(* CoDeSys 2.3 export: CODESYSEXPORT22_2.EXP *)

(* POU MAIN, ST *)
PROGRAM MAIN
(*Main program for application. Uses PackML state model to control the execution of the application*)
VAR
	tonStarting				: TON;
	rsEmergencyClear	: RS;	(*RS - flip-flop for Emergency clear info*)
END_VAR
(* ****** Section 1: Initialisations and default values. Initial conditions for variables on every PLC cycle*)
(*Default values*)
fbStateModel.bSC := FALSE;
(*System resets*)

(* ****** Section 2: Actions in your program without considering the Control Mode. I.e. actions are performed same way indenpendent on
current Control Mode selection.*)
(*Mode independent state actions. Change / Add / Remove states according your need*)
CASE fbStateModel.eState OF
eSt_Aborting:
	(* One can make specific actions in case of specific Mode-State combination.
	   One can also consider to call a specific program when in specific Mode-State combination*)
	actAborting;
	fbStateModel.bSC := TRUE;		(*MODIFY*)
eSt_Clearing:
	fbStateModel.bSC := TRUE;		(*MODIFY*)
eSt_Resetting:
	fbStateModel.bSC := TRUE;
eSt_Holding:
	fbStateModel.bSC := TRUE;		(*MODIFY*)
eSt_UnHolding:
	fbStateModel.bSC := TRUE;		(*MODIFY*)
eSt_Suspending:
	fbStateModel.bSC := TRUE;		(*MODIFY*)
eSt_Unsuspending:
	fbStateModel.bSC := TRUE;		(*MODIFY*)
END_CASE;

(* ****** Section 3: Actions in your program which are Control Mode specific. Two nested case structures where outer one selects the
control mode and inner the PackML state. In order to avoid conflicts, it would be better to process each PackML state either in Section 2 
or Section 3, but not in both. *)
(*Execution mode related state actions. Change / Add / Remove mode and states according your need*)
CASE fbStateModel.eMode OF
(*MODE: MANUAL*)
eMode_Manual:
	(* ****** Section 3.1: PackML state based processing actions when Control Mode is Manual.*)
	CASE fbStateModel.eState OF
	eSt_Starting:
		IF IPressureApplied THEN
			fbStateModel.bSC := TRUE;			(*MODIFY*)
		END_IF
	eSt_Stopping:
		fbStateModel.bSC := TRUE;			(*MODIFY*)
	END_CASE;

(*MODE: AUTOMATIC*)
eMode_Automatic:
	(* ****** Section 3.2: PackML state based processing actions when Control Mode is Automatic.*)
	CASE fbStateModel.eState OF
	eSt_Idle:
		tonStarting(IN:=FALSE , PT:= , Q=> , ET=> );	(*MODIFY*)
	eSt_Starting:
		(* tonStarting(IN:=TRUE , PT:=T#2s , Q=> , ET=> );
		fbStateModel.bSC := tonStarting.Q; *)
		IF IPressureApplied THEN
			bDriveEnabled := TRUE;
			PRG_Initialisation(bReset:= , bExecute:= TRUE , bDone=> );
		END_IF

		IF PRG_Initialisation.bDone THEN
			PRG_Initialisation(bReset:= , bExecute:= FALSE , bDone=> );
			fbStateModel.bSC := TRUE;
		END_IF
	eSt_Completing:
		fbStateModel.bSC := TRUE;					(*MODIFY*)
	eSt_Completed:
		;
	END_CASE;

(* ****** Section 4: Grouping PackML states for calling Programs or FB instances.
This is to avoid repetition inside above case structure in Section 3. With IF clause setting lower (and upper) state limits we can filter out the states when we want to call 
specific programs. The order of states is defined in Tab:Data types > E_PackMLState. eSt_Aborting is lowest and eSt_Completed is highest.
Here we filter calling programs, only when we are in higher states than Stopped. 
This can be pulled out as completely separated section, like in PackML_StateModel_v2-2.pro project. There is inside IF again CASE which process each Control Mode separately.*)
(*Execution part. Making calls for program if we are on states above Stopped*)
	(*If we are between specific states, make some action or program call*)
	IF  (fbStateModel.eState>eSt_Starting) AND (fbStateModel.eState<=eSt_Completing) THEN
		(*Make here the actions / calls Good place to start with is PRG_Sorting (PRG)*)
		PRG_AutoSort(bExecute:= TRUE , bReset:= , bDone=> , bStopOk=> );
	END_IF;

(*MODE: UNKNOWN*)
ELSE	(*Error*)
	; (*TODO*)
END_CASE;

(* ****** Section 5: Calling the fbStateModel instance.
Here the instance of state model is called and all triggering inputs are set, but bSC (State Completed), which you control in your programs. 
This is indication that your program has  finished certain stage.
- Pay attention where the instance fbStateModel is defined. Do you do it in global variables or e.g. here in PRG_MAIN? Important is to use the 
same instance in all places, so that machine state is unique and shared. Remember, if you have multiple definitions, the PRG_MAIN "hides" 
the global one, and might lead to problems elswhere, when you think you are using the same instance, but actually are not. 
- In case you are using the PackML visualisation (VC_PackMLStates), make sure you connect its placeholder to the very same PackML FB instance.
- The Mask for wIgnoreState is created as following. I use binary base for the value(2#). The lowest bit in the mask corresponds the eSt_Aborting
 in E_PackMLState. The next is eSt_Aborted, and so on. Specific state is ignored and jumped over when it is masked out i.e. ignored by having 1 
in that position. Note that implementation allows this only for selected states. See FB_PackMLStateModel_ST code for further details.*)
(*Calling & Updating the state model*)
(*TODO: Evaluate and change all input conditions according your application needs*)
fbStateModel(
	bResetFB:= ,
	eModeReq:= HMI_uModeReq,
	wIgnoreState := 2#000000,		(*TODO: Which states should be ignodered. Default: 2#000000 or 2#100000. The latter is ignoring Resetting state*)
	bSC:= ,			(*Must not be assigned ANY variable, because fb input is directly operated!!!*)
	bAbort:= NOT (IEmergencyClear  OR  IPressureApplied),
	bClear:= IEmergencyClear,
	bReset:= I_Btn_Start,
	bStart:= I_Btn_Start,
	bHold:= ,
	bUn_Hold:= ,
	bSuspend:= ,
	bUn_Suspend:= ,
	bStop:= I_Btn_Stop ,
	bComplete:= ,
	bAck_Completed:= ,
	eMode=> PLC_uModeCurrent,
	eState=> PLC_uStateCurrent);

(* ****** Section 6: Here we update all outputs according the current state of our PackML model. This allows us to process the in single location.
The control of outputs is bind to state, not e.g. to inputs. The inputs are the one driving the PackML model forward. Again CASE structure can be used.*)
(*Call for HMI and UI update*)
(*PRG_Drive_Link()*);
HMI_and_UI_Update;
END_PROGRAM
ACTION actAborting:
bDriveEnabled := FALSE;
PRG_Sorting(bReset:=TRUE , bExecute:= FALSE);
END_ACTION
ACTION HMI_and_UI_Update:
(*Simulate emergency stop circuitry*)
rsEmergencyClear(
	SET:= I_Btn_Reset,
	RESET1:= I_Btn_EStop ,
	Q1=> IEmergencyClear);

(*HMI Update*)
PRG_Blinking (bSign4Hz=> , bSign2Hz=> , bSign1Hz=> , bSign0_5Hz=> );
(*Init values*)
O_Light_BeaconRed := FALSE;

(*OLight_Start :=  (fbStateModel.eState >= eSt_Resetting) AND (fbStateModel.eState < eSt_Completed);*)
CASE fbStateModel.eState OF
eSt_Aborting, eSt_Aborted:
	O_Light_BeaconRed := PRG_Blinking.bSign1Hz;
eSt_Clearing:
	O_Light_BeaconRed := PRG_Blinking.bSign0_5Hz;
eSt_Stopped, eSt_Completed:
	O_Light_BeaconRed := TRUE;
eSt_Starting:
	;
END_CASE;
END_ACTION

(* POU Programs/PRG_Initialisation, SFC *)
PROGRAM PRG_Initialisation
(*Template program for system initialisation*)
VAR_INPUT
	bReset	: BOOL := FALSE;	(*Reseting the SFC*)
	bExecute	: BOOL;			(*Executes PRG*)
END_VAR
VAR_OUTPUT
	bDone		: BOOL;		(*Program operations done*)
END_VAR
VAR
(* -------------INTERNAL-------------------*)
	tonMoveDelay		: TON;
	tMoveDelay		: TIME := T#1s;
	bInitDone			: BOOL:=FALSE;	(*Initialisation done*)
	bGatesClosed	: BOOL:=FALSE;	(*Initialisation done*)
	bActuRetracted	: BOOL:=FALSE;
	bDriveAtLoading	: BOOL:=FALSE;

(*System variables. See SFC-flags: http://infosys.beckhoff.com/content/1033/tcplccontrol/html/tcplcctrl_editorsfc.htm?id=24319#SFC-Flags*)
	SFCReset		: BOOL := FALSE;	(*For reseting the SFC*)
END_VAR
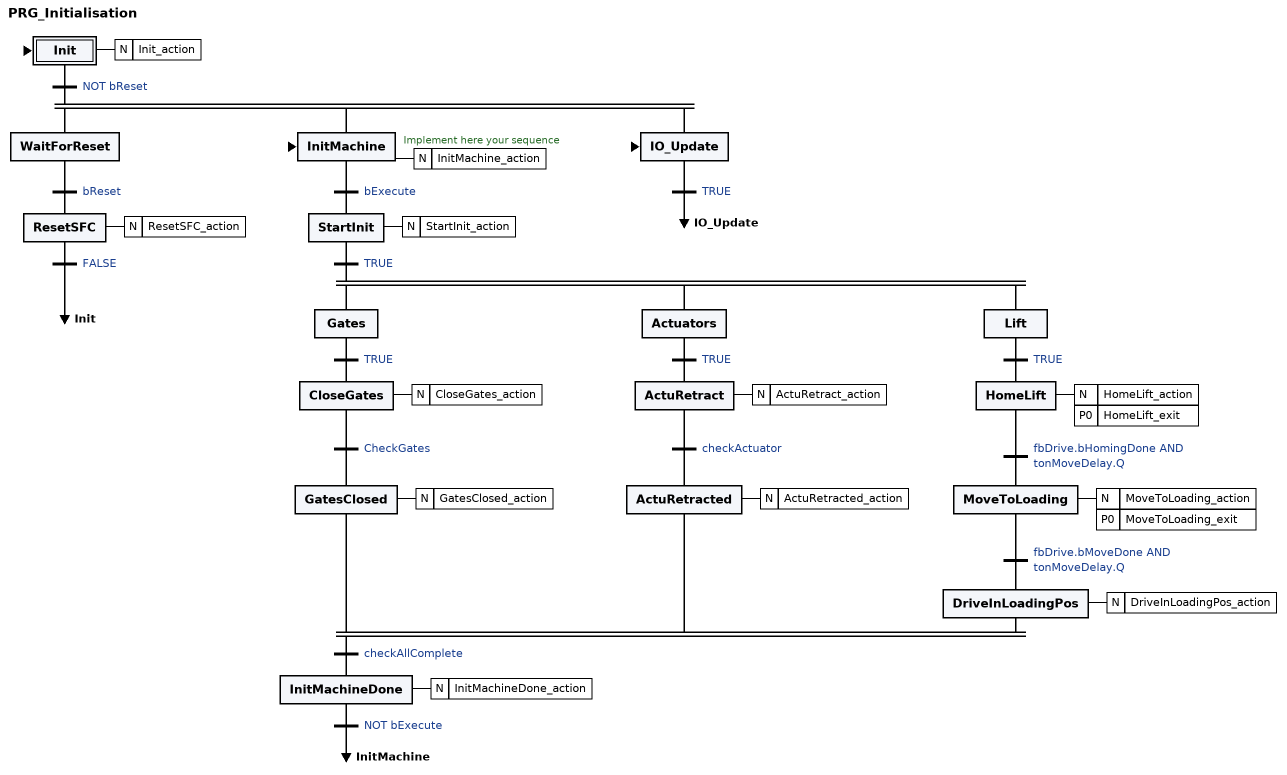
INITIAL_STEP Init:
	Init_action(N);
END_STEP
TRANSITION FROM Init TO (WaitForReset, InitMachine, IO_Update) := NOT bReset;
END_TRANSITION
STEP WaitForReset:
END_STEP
TRANSITION FROM WaitForReset TO ResetSFC := bReset;
END_TRANSITION
STEP ResetSFC:
	ResetSFC_action(N);
END_STEP
TRANSITION FROM ResetSFC TO Init := FALSE;
END_TRANSITION
STEP InitMachine: (* Implement here your sequence *)
	InitMachine_action(N);
END_STEP
TRANSITION FROM InitMachine TO StartInit := bExecute;
END_TRANSITION
STEP StartInit:
	StartInit_action(N);
END_STEP
TRANSITION FROM StartInit TO (Gates, Actuators, Lift) := TRUE;
END_TRANSITION
STEP Gates:
END_STEP
TRANSITION FROM Gates TO CloseGates := TRUE;
END_TRANSITION
STEP CloseGates:
	CloseGates_action(N);
END_STEP
TRANSITION FROM CloseGates TO GatesClosed := CheckGates;
END_TRANSITION
STEP GatesClosed:
	GatesClosed_action(N);
END_STEP
STEP Actuators:
END_STEP
TRANSITION FROM Actuators TO ActuRetract := TRUE;
END_TRANSITION
STEP ActuRetract:
	ActuRetract_action(N);
END_STEP
TRANSITION FROM ActuRetract TO ActuRetracted := checkActuator;
END_TRANSITION
STEP ActuRetracted:
	ActuRetracted_action(N);
END_STEP
STEP Lift:
END_STEP
TRANSITION FROM Lift TO HomeLift := TRUE;
END_TRANSITION
STEP HomeLift:
	HomeLift_action(N);
	HomeLift_exit(P0);
END_STEP
TRANSITION FROM HomeLift TO MoveToLoading := fbDrive.bHomingDone AND tonMoveDelay.Q;
END_TRANSITION
STEP MoveToLoading:
	MoveToLoading_action(N);
	MoveToLoading_exit(P0);
END_STEP
TRANSITION FROM MoveToLoading TO DriveInLoadingPos := fbDrive.bMoveDone AND tonMoveDelay.Q;
END_TRANSITION
STEP DriveInLoadingPos:
	DriveInLoadingPos_action(N);
END_STEP
TRANSITION FROM (GatesClosed, ActuRetracted, DriveInLoadingPos) TO InitMachineDone := checkAllComplete;
END_TRANSITION
STEP InitMachineDone:
	InitMachineDone_action(N);
END_STEP
TRANSITION FROM InitMachineDone TO InitMachine := NOT bExecute;
END_TRANSITION
STEP IO_Update:
END_STEP
TRANSITION FROM IO_Update TO IO_Update := TRUE;
END_TRANSITION

ACTION Init_action:
(*Clear Reset SFC*)
SFCReset:= FALSE;
bDone := FALSE;
END_ACTION

ACTION ResetSFC_action:
(*Reset SFC*)
SFCReset:=TRUE;
END_ACTION

ACTION InitMachine_action:
(*Do some actions...

Sulje kaikki portit ... JA tarkista Steppiä seuraavassa transitioehdossa, että kaikki portit ovat kiinni
Close all gates.... and check in following transition that ALL gates are closed*)

;
END_ACTION

ACTION StartInit_action:
bDone := FALSE;
END_ACTION

ACTION CloseGates_action:
OGateUp		:= FALSE;
OGateMid		:= FALSE;
OGateLow		:= FALSE;
OSorterGate	:= FALSE;
END_ACTION

ACTION GatesClosed_action:
bGatesClosed := TRUE;
END_ACTION

ACTION ActuRetract_action:
OSorterLift	 := FALSE;
OEjector	 := FALSE;
END_ACTION

ACTION ActuRetracted_action:
bActuRetracted := TRUE;
END_ACTION

ACTION HomeLift_action:
fbDrive.bStart := TRUE;
tonMoveDelay(IN:=TRUE , PT:= tMoveDelay);
END_ACTION

ACTION HomeLift_exit:
fbDrive.bStart:= FALSE;
tonMoveDelay(IN:=FALSE);
END_ACTION

ACTION MoveToLoading_action:
fbDrive.wTarget := GPOS_LOADING;
fbDrive.bStart:= TRUE;
tonMoveDelay(IN:=TRUE , PT:= tMoveDelay);
END_ACTION

ACTION MoveToLoading_exit:
fbDrive.bStart:= FALSE;
tonMoveDelay(IN:=FALSE);
END_ACTION

ACTION DriveInLoadingPos_action:
bDriveAtLoading := TRUE;
END_ACTION

ACTION InitMachineDone_action:
bDone := TRUE;
END_ACTION

TRANSITION CheckGates:
_FBD_ (* Function Block Diagram *)
NETWORK 1
	AND(IGateClosedUp, IGateClosedMid, IGateClosedLow, ISorterGateClosed)
_END_FBD_
END_TRANSITION

TRANSITION checkActuator:
_FBD_ (* Function Block Diagram *)
NETWORK 1
	AND(ISorterLiftDown, NOT OEjector)
_END_FBD_
END_TRANSITION

TRANSITION checkAllComplete:
_FBD_ (* Function Block Diagram *)
NETWORK 1
	AND(bGatesClosed, bActuRetracted, bDriveAtLoading)
_END_FBD_
END_TRANSITION
END_PROGRAM

(* POU Programs/PRG_AutoSort, ST *)
PROGRAM PRG_AutoSort
VAR_INPUT
	bExecute	: BOOL;
	bReset	: BOOL := FALSE;
END_VAR
VAR_OUTPUT
	bDone		: BOOL;		(*Program operations done*)
	bStopOk    : BOOL;
END_VAR
VAR
	fbSorter	: FB_Sorter;
	fbLift		: FB_Lift;
	bBatchComplete  : BOOL := FALSE;
END_VAR
actUpdateIO;
actCheckAllOkStop;

CASE fbStateModel.eState OF
	eSt_Idle:
		fbStateModel.bComplete  := FALSE;
		fbStateModel.bSC 		:= TRUE;
	eSt_Resetting:
		fbStateModel.bSC := TRUE;
	eSt_Stopping:
		fbStateModel.bStop := FALSE;

		IF  bStopOk THEN
			fbStateModel.bSC := TRUE;
		END_IF
	eSt_Execute:
		fbSorter (bEnable :=  TRUE , bReset := FALSE);
		fbLift(bEnable :=  TRUE , bReset := FALSE);
		IF bBatchComplete  THEN
			fbStateModel.bComplete := TRUE;
		END_IF

	eSt_Completing:
		fbStateModel.bComplete := FALSE;
		IF bStopOK THEN
			fbStateModel.bSC := TRUE;
		END_IF

	eSt_Unsuspending:
		fbStateModel.bSC := TRUE;

	eSt_Suspending:
		fbStateModel.bSuspend := FALSE;
		fbStateModel.bSC := TRUE;

END_CASE
END_PROGRAM
ACTION actCheckAllOKStop:
IF fbSorter.bStopOK AND  fbLift.bStopOK THEN
	bStopOK := TRUE;
ELSE
	bStopOK := FALSE;
END_IF
END_ACTION
ACTION actUpdateIO:
fbSorter (
	bReset:= ,
	bEnable:= bExecute,
	I_SensorOpt:= ISensorOpt ,
	I_SensorInd:= ISensorInd,
	I_SorterLiftUp:= ISorterLiftUp ,
	I_SorterLiftDown:= ISorterLiftDown,
	hiRdyToReceive_FromDS:= fbLift.hoReadyToRecieve_ToUS ,
	hiBallAvail_FromUS:= ,
	bStopOK=> ,
	bBallLoaded=> ,
	bCurBallMetal=> ,
	O_SorterGate=> OSorterGate ,
	O_SorterLift=> OSorterLift ,
	hoBallAvail_ToDS=> ,
	hoReadyToRecieve_ToUS=> );

fbLift (
	bReset:= ,
	bEnable:= bExecute,
	I_LimitUp:= ILimitUp  ,
	I_LimitLow:= ILimitLow,
	I_WaitingBallMetal:= fbSorter.bCurBallMetal  ,
	I_SenColourYellow:= ISenColourYellow ,
	I_SenColourBlue:= ISenColourBlue ,
	I_SenColourGreen:= ISenColourGreen,
	I_SenColourRed:= ISenColourRed ,
	hiRdyToReceive_FromDS:= ,
	hiBallAvail_FromUS:= fbSorter.hoBallAvail_ToDS ,
	bStopOK=> ,
	bBallLoaded=> , 
	bCurBallMetal=> , 
	O_Ejector=> OEjector ,
	hoBallAvail_ToDS=> , 
	hoReadyToRecieve_ToUS=> );
END_ACTION

(* POU FBs/FB_Sorter, SFC *)
FUNCTION_BLOCK FB_Sorter
VAR_INPUT
	bReset			: BOOL;	(*Reset Request*)
	bEnable			: BOOL;
	I_SensorOpt		: BOOL;
	I_SensorInd		: BOOL;
	I_SorterLiftUp		: BOOL;
	I_SorterLiftDown	: BOOL;

	(*SMEMA Handshake Inputs*)
	hiRdyToReceive_FromDS	: BOOL;
	hiBallAvail_FromUS			: BOOL;
END_VAR
VAR_OUTPUT
	bStopOK			: BOOL;
	bBallLoaded		: BOOL;
	bCurBallMetal		: BOOL;
	O_SorterGate		: BOOL;
	O_SorterLift		: BOOL;

	(*SMEMA Handshake Outputs*)
	hoBallAvail_ToDS				: BOOL;
	hoReadyToRecieve_ToUS	: BOOL;
END_VAR
VAR
	tTransferDelay: TIME := T#4s;
	tMoveDelay	: TIME := T#2s;
	fbDelay		: FB_Wait;
	bLocalReset	: BOOL;	(*Performs local reset*)
	SFCReset 	: BOOL;	(*Resets the execution of SFC to init once this SFCFlag is set true *)
END_VAR
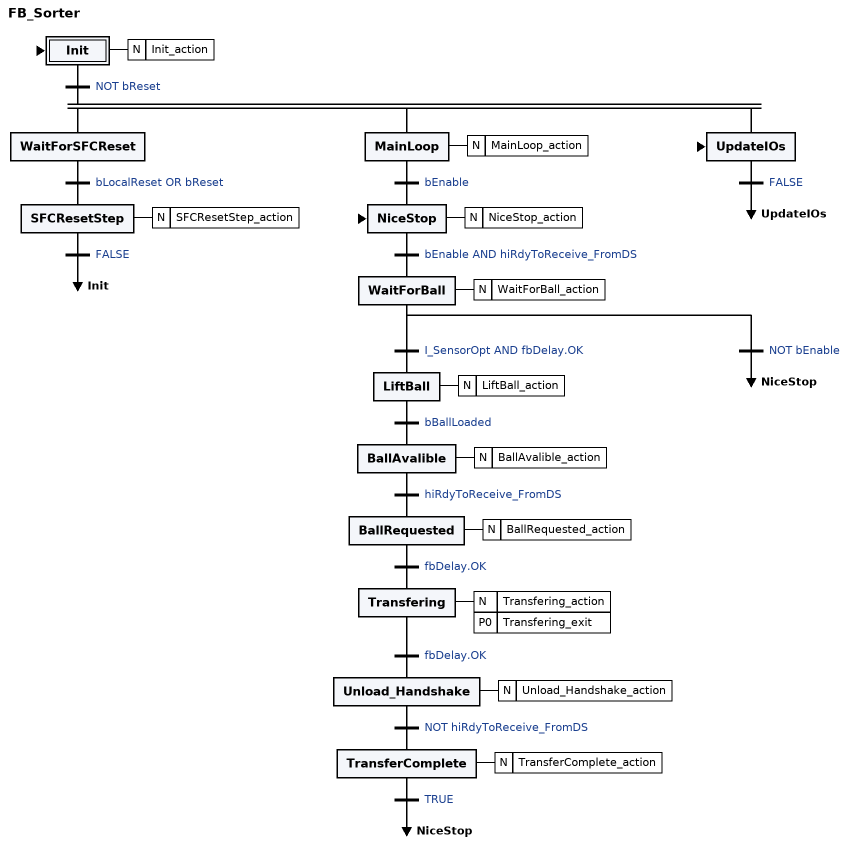
INITIAL_STEP Init:
	Init_action(N);
END_STEP
TRANSITION FROM Init TO (WaitForSFCReset, MainLoop, UpdateIOs) := NOT bReset;
END_TRANSITION
STEP WaitForSFCReset:
END_STEP
TRANSITION FROM WaitForSFCReset TO SFCResetStep := bLocalReset OR bReset;
END_TRANSITION
STEP MainLoop:
	MainLoop_action(N);
END_STEP
TRANSITION FROM MainLoop TO NiceStop := bEnable;
END_TRANSITION
STEP NiceStop:
	NiceStop_action(N);
END_STEP
TRANSITION FROM NiceStop TO WaitForBall := bEnable AND hiRdyToReceive_FromDS;
END_TRANSITION
STEP WaitForBall:
	WaitForBall_action(N);
END_STEP
TRANSITION FROM WaitForBall TO LiftBall := I_SensorOpt AND fbDelay.OK;
END_TRANSITION
TRANSITION FROM WaitForBall TO NiceStop := NOT bEnable;
END_TRANSITION
STEP LiftBall:
	LiftBall_action(N);
END_STEP
TRANSITION FROM LiftBall TO BallAvalible := bBallLoaded;
END_TRANSITION
STEP BallAvalible:
	BallAvalible_action(N);
END_STEP
TRANSITION FROM BallAvalible TO BallRequested := hiRdyToReceive_FromDS;
END_TRANSITION
STEP BallRequested:
	BallRequested_action(N);
END_STEP
TRANSITION FROM BallRequested TO Transfering := fbDelay.OK;
END_TRANSITION
STEP Transfering:
	Transfering_action(N);
	Transfering_exit(P0);
END_STEP
TRANSITION FROM Transfering TO Unload_Handshake := fbDelay.OK;
END_TRANSITION
STEP Unload_Handshake:
	Unload_Handshake_action(N);
END_STEP
TRANSITION FROM Unload_Handshake TO TransferComplete := NOT hiRdyToReceive_FromDS;
END_TRANSITION
STEP TransferComplete:
	TransferComplete_action(N);
END_STEP
TRANSITION FROM TransferComplete TO NiceStop := TRUE;
END_TRANSITION
STEP UpdateIOs:
END_STEP
TRANSITION FROM UpdateIOs TO UpdateIOs := FALSE;
END_TRANSITION
STEP SFCResetStep:
	SFCResetStep_action(N);
END_STEP
TRANSITION FROM SFCResetStep TO Init := FALSE;
END_TRANSITION

ACTION Init_action:
SFCReset := FALSE;
bLocalReset	:= FALSE;
bStopOK := FALSE;
END_ACTION

ACTION MainLoop_action:
hoBallAvail_ToDS			  := FALSE;
hoReadyToRecieve_ToUS := FALSE;
END_ACTION

ACTION NiceStop_action:
bBallLoaded 				  := FALSE;
bStopOK					  := TRUE;
hoBallAvail_ToDS			  := FALSE;
hoReadyToRecieve_ToUS := FALSE;
END_ACTION

ACTION WaitForBall_action:
fbDelay(IN_TIME:=tMoveDelay);
(* Move Lift Down *)
O_SorterLift := FALSE;
END_ACTION

ACTION LiftBall_action:
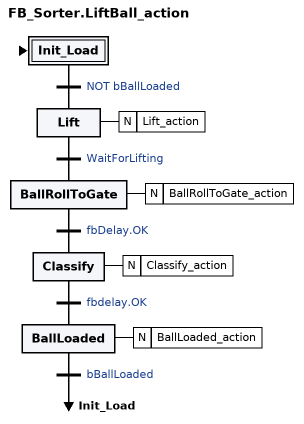
INITIAL_STEP Init_Load:
END_STEP
TRANSITION FROM Init_Load TO Lift := NOT bBallLoaded;
END_TRANSITION
STEP Lift:
	Lift_action(N);
END_STEP
TRANSITION FROM Lift TO BallRollToGate := WaitForLifting;
END_TRANSITION
STEP BallRollToGate:
	BallRollToGate_action(N);
END_STEP
TRANSITION FROM BallRollToGate TO Classify := fbDelay.OK;
END_TRANSITION
STEP Classify:
	Classify_action(N);
END_STEP
TRANSITION FROM Classify TO BallLoaded := fbdelay.OK;
END_TRANSITION
STEP BallLoaded:
	BallLoaded_action(N);
END_STEP
TRANSITION FROM BallLoaded TO Init_Load := bBallLoaded;
END_TRANSITION

ACTION Lift_action:
O_SorterLift := TRUE;
fbDelay(IN_TIME:=tMoveDelay);
END_ACTION

ACTION BallRollToGate_action:
fbDelay(IN_TIME:=tMoveDelay);
END_ACTION

ACTION Classify_action:
fbDelay(IN_TIME:=tMoveDelay);
IF I_SensorInd THEN
	bCurBallMetal := FALSE;
ELSE
	bCurBallMetal := TRUE;
END_IF
END_ACTION

ACTION BallLoaded_action:
bBallLoaded := TRUE;
END_ACTION

TRANSITION WaitForLifting:
_FBD_ (* Function Block Diagram *)
NETWORK 1
	AND(I_SorterLiftUp, fbDelay.OK, NOT I_SensorOpt)
_END_FBD_
END_TRANSITION
END_ACTION

ACTION BallAvalible_action:
hoBallAvail_ToDS := TRUE;
END_ACTION

ACTION BallRequested_action:
fbDelay(IN_TIME:=tMoveDelay);
END_ACTION

ACTION Transfering_action:
O_SorterGate := TRUE;
fbDelay(IN_TIME:=tTransferDelay);
END_ACTION

ACTION Transfering_exit:
O_SorterGate := FALSE;
END_ACTION

ACTION Unload_Handshake_action:
hoBallAvail_ToDS := FALSE;
END_ACTION

ACTION TransferComplete_action:
bBallLoaded := FALSE;
END_ACTION

ACTION SFCResetStep_action:
SFCReset := TRUE;
END_ACTION
END_FUNCTION_BLOCK

(* POU FBs/FB_Lift, SFC *)
FUNCTION_BLOCK FB_Lift
VAR_INPUT
	bReset			 : BOOL;	(*Reset Request*)
	bEnable			 : BOOL;
	I_LimitUp 			 : BOOL;
	I_LimitLow 	        : BOOL;
	I_WaitingBallMetal : BOOL;

	(* ColourSensor *)
	I_SenColourYellow		:BOOL;	(*Colour sensor In1 - Yellow*)
	I_SenColourBlue		:BOOL;	(*Colour sensor In2 - Blue*)
	I_SenColourGreen		:BOOL;	(*Colour sensor In3 - Green*)
	I_SenColourRed		:BOOL;	(*Colour sensor In4 - Red*)

	(*SMEMA Handshake Inputs*)
	hiRdyToReceive_FromDS	: BOOL;
	hiBallAvail_FromUS			: BOOL;
END_VAR
VAR_OUTPUT
	bStopOK		: BOOL;
	bBallLoaded	: BOOL;
	bCurBallMetal	: BOOL;
	bCurrentBall 	: E_BallColour := NoColour;

	O_Ejector		:BOOL;

	(*SMEMA Handshake Outputs*)
	hoBallAvail_ToDS				: BOOL;
	hoReadyToRecieve_ToUS	: BOOL;
END_VAR
VAR
	bBallRequested : BOOL := FALSE;
	fbTransferBall	:FB_TransferBall;

	fbDelay		: FB_Wait;
	tonMoveDelay	: TON;
	tonSensorDelay	: TON;
	tTransferDelay: TIME := T#4s;
	tMoveDelay	: TIME := T#4s;
	tSensorDelay	: TIME := T#2s;
	bLocalReset	: BOOL;	(*Performs local reset*)
	SFCReset 	: BOOL;	(*Resets the execution of SFC to init once this SFCFlag is set true *)
END_VAR
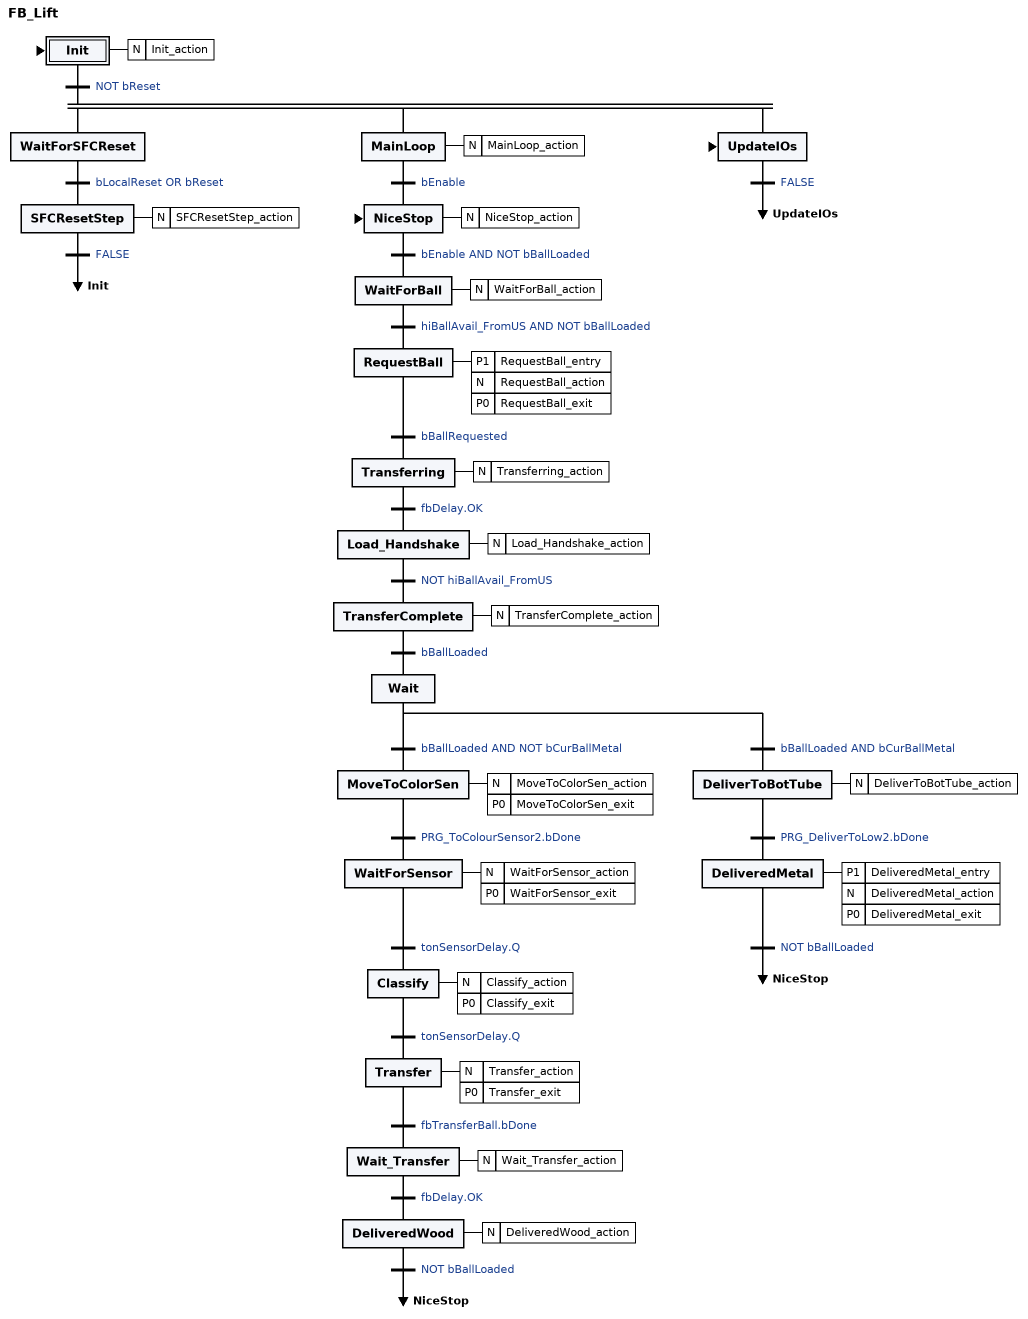
INITIAL_STEP Init:
	Init_action(N);
END_STEP
TRANSITION FROM Init TO (WaitForSFCReset, MainLoop, UpdateIOs) := NOT bReset;
END_TRANSITION
STEP WaitForSFCReset:
END_STEP
TRANSITION FROM WaitForSFCReset TO SFCResetStep := bLocalReset OR bReset;
END_TRANSITION
STEP MainLoop:
	MainLoop_action(N);
END_STEP
TRANSITION FROM MainLoop TO NiceStop := bEnable;
END_TRANSITION
STEP NiceStop:
	NiceStop_action(N);
END_STEP
TRANSITION FROM NiceStop TO WaitForBall := bEnable AND NOT bBallLoaded;
END_TRANSITION
STEP WaitForBall:
	WaitForBall_action(N);
END_STEP
TRANSITION FROM WaitForBall TO RequestBall := hiBallAvail_FromUS AND NOT bBallLoaded;
END_TRANSITION
STEP RequestBall:
	RequestBall_entry(P1);
	RequestBall_action(N);
	RequestBall_exit(P0);
END_STEP
TRANSITION FROM RequestBall TO Transferring := bBallRequested;
END_TRANSITION
STEP Transferring:
	Transferring_action(N);
END_STEP
TRANSITION FROM Transferring TO Load_Handshake := fbDelay.OK;
END_TRANSITION
STEP Load_Handshake:
	Load_Handshake_action(N);
END_STEP
TRANSITION FROM Load_Handshake TO TransferComplete := NOT hiBallAvail_FromUS;
END_TRANSITION
STEP TransferComplete:
	TransferComplete_action(N);
END_STEP
TRANSITION FROM TransferComplete TO Wait := bBallLoaded;
END_TRANSITION
STEP Wait:
END_STEP
TRANSITION FROM Wait TO MoveToColorSen := bBallLoaded AND NOT bCurBallMetal;
END_TRANSITION
TRANSITION FROM Wait TO DeliverToBotTube := bBallLoaded AND bCurBallMetal;
END_TRANSITION
STEP MoveToColorSen:
	MoveToColorSen_action(N);
	MoveToColorSen_exit(P0);
END_STEP
TRANSITION FROM MoveToColorSen TO WaitForSensor := PRG_ToColourSensor2.bDone;
END_TRANSITION
STEP WaitForSensor:
	WaitForSensor_action(N);
	WaitForSensor_exit(P0);
END_STEP
TRANSITION FROM WaitForSensor TO Classify := tonSensorDelay.Q;
END_TRANSITION
STEP Classify:
	Classify_action(N);
	Classify_exit(P0);
END_STEP
TRANSITION FROM Classify TO Transfer := tonSensorDelay.Q;
END_TRANSITION
STEP Transfer:
	Transfer_action(N);
	Transfer_exit(P0);
END_STEP
TRANSITION FROM Transfer TO Wait_Transfer := fbTransferBall.bDone;
END_TRANSITION
STEP Wait_Transfer:
	Wait_Transfer_action(N);
END_STEP
TRANSITION FROM Wait_Transfer TO DeliveredWood := fbDelay.OK;
END_TRANSITION
STEP DeliveredWood:
	DeliveredWood_action(N);
END_STEP
TRANSITION FROM DeliveredWood TO NiceStop := NOT bBallLoaded;
END_TRANSITION
STEP DeliverToBotTube:
	DeliverToBotTube_action(N);
END_STEP
TRANSITION FROM DeliverToBotTube TO DeliveredMetal := PRG_DeliverToLow2.bDone;
END_TRANSITION
STEP DeliveredMetal:
	DeliveredMetal_entry(P1);
	DeliveredMetal_action(N);
	DeliveredMetal_exit(P0);
END_STEP
TRANSITION FROM DeliveredMetal TO NiceStop := NOT bBallLoaded;
END_TRANSITION
STEP UpdateIOs:
END_STEP
TRANSITION FROM UpdateIOs TO UpdateIOs := FALSE;
END_TRANSITION
STEP SFCResetStep:
	SFCResetStep_action(N);
END_STEP
TRANSITION FROM SFCResetStep TO Init := FALSE;
END_TRANSITION

ACTION Init_action:
SFCReset := FALSE;
bLocalReset	:= FALSE;
END_ACTION

ACTION MainLoop_action:
hoBallAvail_ToDS			  := FALSE;
hoReadyToRecieve_ToUS := FALSE;
END_ACTION

ACTION NiceStop_action:
bStopOK	  	:= TRUE;
bCurrentBall	:= NoColour;
END_ACTION

ACTION WaitForBall_action:
bBallLoaded := FALSE;
hoReadyToRecieve_ToUS := TRUE;
END_ACTION

ACTION RequestBall_entry:
bStopOK := FALSE;
END_ACTION

ACTION RequestBall_action:
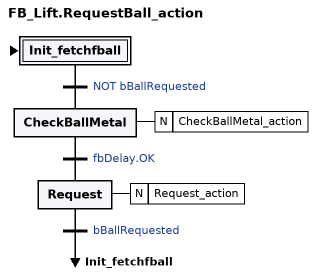
INITIAL_STEP Init_fetchfball:
END_STEP
TRANSITION FROM Init_fetchfball TO CheckBallMetal := NOT bBallRequested;
END_TRANSITION
STEP CheckBallMetal:
	CheckBallMetal_action(N);
END_STEP
TRANSITION FROM CheckBallMetal TO Request := fbDelay.OK;
END_TRANSITION
STEP Request:
	Request_action(N);
END_STEP
TRANSITION FROM Request TO Init_fetchfball := bBallRequested;
END_TRANSITION

ACTION CheckBallMetal_action:
bCurBallMetal	 := I_WaitingBallMetal;
fbDelay(IN_TIME:=T#2s);
END_ACTION

ACTION Request_action:
hoReadyToRecieve_ToUS := TRUE;
bBallRequested := TRUE;
END_ACTION
END_ACTION

ACTION RequestBall_exit:
bBallRequested := FALSE;
END_ACTION

ACTION Transferring_action:
fbDelay(IN_TIME:=tTransferDelay);
END_ACTION

ACTION Load_Handshake_action:
hoReadyToRecieve_ToUS := FALSE;
END_ACTION

ACTION TransferComplete_action:
bBallLoaded := TRUE;
END_ACTION

ACTION MoveToColorSen_action:
PRG_ToColourSensor2(bExecute:=TRUE , bDone=> );
END_ACTION

ACTION MoveToColorSen_exit:
PRG_ToColourSensor2( bExecute:=FALSE);
END_ACTION

ACTION WaitForSensor_action:
tonSensorDelay(IN:=TRUE , PT:= tSensorDelay);
END_ACTION

ACTION WaitForSensor_exit:
tonSensorDelay(IN:=FALSE);
END_ACTION

ACTION Classify_action:
tonSensorDelay(IN:=TRUE , PT:= tSensorDelay);
IF I_SenColourYellow THEN
	bCurrentBall := Yellow;
ELSIF  I_SenColourBlue THEN
	bCurrentBall := Blue;
ELSIF  I_SenColourRed THEN
	bCurrentBall := Red;
ELSE
	bCurrentBall := NoColour;
END_IF
END_ACTION

ACTION Classify_exit:
tonSensorDelay(IN:=FALSE);
END_ACTION

ACTION Transfer_action:
fbTransferBall(bExecute:= TRUE , bBallToTransfer:= bCurrentBall, bDone=> );
END_ACTION

ACTION Transfer_exit:
fbTransferBall(bExecute:= FALSE);
END_ACTION

ACTION Wait_Transfer_action:
fbDelay(IN_TIME:=tMoveDelay);
END_ACTION

ACTION DeliveredWood_action:
bBallLoaded := FALSE;
bCurrentBall := NoColour;
END_ACTION

ACTION DeliverToBotTube_action:
PRG_DeliverToLow2(bExecute:=TRUE ,  bDone=> );
END_ACTION

ACTION DeliveredMetal_entry:
bBallLoaded := FALSE;
PRG_DeliverToLow(bReset:=FALSE , bExecute:=FALSE ,  bDone=> );
END_ACTION

ACTION DeliveredMetal_action:
bBallLoaded := FALSE;
END_ACTION

ACTION DeliveredMetal_exit:
PRG_DeliverToLow(bReset:=FALSE , bExecute:=FALSE ,  bDone=> );
END_ACTION

ACTION SFCResetStep_action:
SFCReset := TRUE;
END_ACTION
END_FUNCTION_BLOCK

(* POU FBs/FB_TransferBall, ST *)
FUNCTION_BLOCK FB_TransferBall
VAR_INPUT
	bExecute			: BOOL;	(*enable and run*)
	bBallToTransfer 	: E_BallColour;
END_VAR
VAR_OUTPUT
	bDone			: BOOL;
	bActDone		: BOOL := FALSE;
END_VAR
VAR
	tonMoveDelay	: TON;
	tonEjectDelay	: TON;
	tMoveDelay	: TIME := T#4s;
	tEjectorDelay	: TIME := T#2s;
END_VAR
IF bExecute THEN
	CASE bBallToTransfer OF
		Yellow:
			PRG_DeliverToUp2( bExecute:= TRUE , bDone=> );
				bDone	:= FALSE;
				IF PRG_DeliverToUp2.bDone THEN
					PRG_DeliverToUp2(bExecute:=FALSE);
					bDone	:= TRUE;
				END_IF
		Blue:
			PRG_DeliverToMid2( bExecute:= TRUE, bDone=> );
				bDone	:= FALSE;
				IF PRG_DeliverToMid2.bDone THEN
					PRG_DeliverToMid2(bExecute:=FALSE);
					bDone	:= TRUE;
				END_IF
		Red:
			PRG_DeliverToGarbage2( bExecute:= TRUE, bDone=> );
				bDone	:= FALSE;
				IF PRG_DeliverToGarbage2.bDone THEN
					PRG_DeliverToGarbage2( bExecute:=FALSE);
					bDone	:= TRUE;
				END_IF
	ELSE
		PRG_DeliverToMid2(bExecute:=FALSE);
		PRG_DeliverToUp2(bExecute:=FALSE);
		PRG_DeliverToGarbage2( bExecute:=FALSE);
		bDone	:= FALSE;
	END_CASE
ELSE
	bDone := FALSE;
END_IF
END_FUNCTION_BLOCK

(* POU Processes/PRG_DeliverToUp2, SFC *)
PROGRAM PRG_DeliverToUp2
VAR_INPUT
	bExecute: BOOL;
END_VAR
VAR_INPUT
	bDone: BOOL;
END_VAR
VAR
	tonMoveDelay	: TON;
	tonEjectDelay	: TON;
	tMoveDelay	: TIME := T#3s;
	tEjectorDelay	: TIME := T#3s;
END_VAR
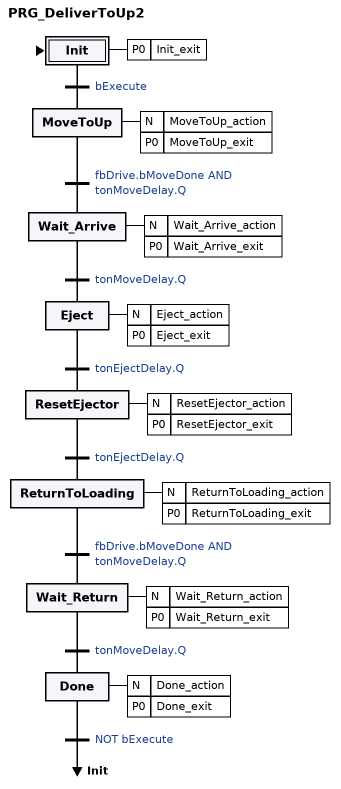
INITIAL_STEP Init:
	Init_exit(P0);
END_STEP
TRANSITION FROM Init TO MoveToUp := bExecute;
END_TRANSITION
STEP MoveToUp:
	MoveToUp_action(N);
	MoveToUp_exit(P0);
END_STEP
TRANSITION FROM MoveToUp TO Wait_Arrive := fbDrive.bMoveDone AND tonMoveDelay.Q;
END_TRANSITION
STEP Wait_Arrive:
	Wait_Arrive_action(N);
	Wait_Arrive_exit(P0);
END_STEP
TRANSITION FROM Wait_Arrive TO Eject := tonMoveDelay.Q;
END_TRANSITION
STEP Eject:
	Eject_action(N);
	Eject_exit(P0);
END_STEP
TRANSITION FROM Eject TO ResetEjector := tonEjectDelay.Q;
END_TRANSITION
STEP ResetEjector:
	ResetEjector_action(N);
	ResetEjector_exit(P0);
END_STEP
TRANSITION FROM ResetEjector TO ReturnToLoading := tonEjectDelay.Q;
END_TRANSITION
STEP ReturnToLoading:
	ReturnToLoading_action(N);
	ReturnToLoading_exit(P0);
END_STEP
TRANSITION FROM ReturnToLoading TO Wait_Return := fbDrive.bMoveDone AND tonMoveDelay.Q;
END_TRANSITION
STEP Wait_Return:
	Wait_Return_action(N);
	Wait_Return_exit(P0);
END_STEP
TRANSITION FROM Wait_Return TO Done := tonMoveDelay.Q;
END_TRANSITION
STEP Done:
	Done_action(N);
	Done_exit(P0);
END_STEP
TRANSITION FROM Done TO Init := NOT bExecute;
END_TRANSITION

ACTION Init_exit:
bDone := FALSE;
END_ACTION

ACTION MoveToUp_action:
fbDrive(
	bEnable:= TRUE,
	bStart:= TRUE,
	wTarget:= GPOS_PIPE_UP);

tonMoveDelay(IN:=TRUE , PT:= tMoveDelay);
END_ACTION

ACTION MoveToUp_exit:
fbDrive(
	bStart:= FALSE);
tonMoveDelay(IN:=FALSE);
END_ACTION

ACTION Wait_Arrive_action:
tonMoveDelay(IN:=TRUE , PT:= tMoveDelay);
END_ACTION

ACTION Wait_Arrive_exit:
tonMoveDelay(IN:=FALSE);
END_ACTION

ACTION Eject_action:
OEjector := TRUE;
tonEjectDelay(IN:=TRUE , PT:= tEjectorDelay);
END_ACTION

ACTION Eject_exit:
tonEjectDelay(IN:=FALSE);
END_ACTION

ACTION ResetEjector_action:
OEjector := FALSE;
tonEjectDelay(IN:=TRUE , PT:= tEjectorDelay);
END_ACTION

ACTION ResetEjector_exit:
tonEjectDelay(IN:=FALSE);
END_ACTION

ACTION ReturnToLoading_action:
fbDrive(
	bEnable:= TRUE,
	bStart:= TRUE,
	wTarget:= GPOS_LOADING);

tonMoveDelay(IN:=TRUE , PT:= tMoveDelay);
END_ACTION

ACTION ReturnToLoading_exit:
fbDrive(
	bStart:= FALSE);

tonMoveDelay(IN:=FALSE);
END_ACTION

ACTION Wait_Return_action:
tonMoveDelay(IN:=TRUE , PT:= tMoveDelay);
END_ACTION

ACTION Wait_Return_exit:
tonMoveDelay(IN:=FALSE);
END_ACTION

ACTION Done_action:
bDone := TRUE;
END_ACTION

ACTION Done_exit:
bDone := FALSE;
END_ACTION
END_PROGRAM

(* POU Processes/PRG_DeliverToMid2, SFC *)
PROGRAM PRG_DeliverToMid2
VAR_INPUT
	bExecute: BOOL;
END_VAR
VAR_INPUT
	bDone: BOOL;
END_VAR
VAR
	tonMoveDelay	: TON;
	tonEjectDelay	: TON;
	tMoveDelay	: TIME := T#3s;
	tEjectorDelay	: TIME := T#3s;
END_VAR
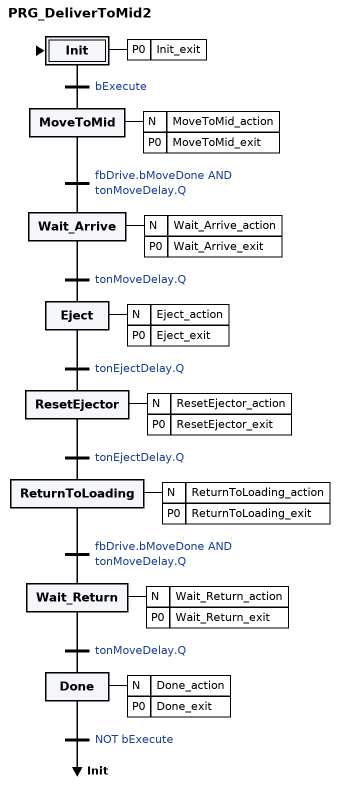
INITIAL_STEP Init:
	Init_exit(P0);
END_STEP
TRANSITION FROM Init TO MoveToMid := bExecute;
END_TRANSITION
STEP MoveToMid:
	MoveToMid_action(N);
	MoveToMid_exit(P0);
END_STEP
TRANSITION FROM MoveToMid TO Wait_Arrive := fbDrive.bMoveDone AND tonMoveDelay.Q;
END_TRANSITION
STEP Wait_Arrive:
	Wait_Arrive_action(N);
	Wait_Arrive_exit(P0);
END_STEP
TRANSITION FROM Wait_Arrive TO Eject := tonMoveDelay.Q;
END_TRANSITION
STEP Eject:
	Eject_action(N);
	Eject_exit(P0);
END_STEP
TRANSITION FROM Eject TO ResetEjector := tonEjectDelay.Q;
END_TRANSITION
STEP ResetEjector:
	ResetEjector_action(N);
	ResetEjector_exit(P0);
END_STEP
TRANSITION FROM ResetEjector TO ReturnToLoading := tonEjectDelay.Q;
END_TRANSITION
STEP ReturnToLoading:
	ReturnToLoading_action(N);
	ReturnToLoading_exit(P0);
END_STEP
TRANSITION FROM ReturnToLoading TO Wait_Return := fbDrive.bMoveDone AND tonMoveDelay.Q;
END_TRANSITION
STEP Wait_Return:
	Wait_Return_action(N);
	Wait_Return_exit(P0);
END_STEP
TRANSITION FROM Wait_Return TO Done := tonMoveDelay.Q;
END_TRANSITION
STEP Done:
	Done_action(N);
	Done_exit(P0);
END_STEP
TRANSITION FROM Done TO Init := NOT bExecute;
END_TRANSITION

ACTION Init_exit:
bDone := FALSE;
END_ACTION

ACTION MoveToMid_action:
fbDrive(
	bEnable:= TRUE,
	bStart:= TRUE,
	wTarget:= GPOS_PIPE_MID);

tonMoveDelay(IN:=TRUE , PT:= tMoveDelay);
END_ACTION

ACTION MoveToMid_exit:
fbDrive(
	bStart:= FALSE);
tonMoveDelay(IN:=FALSE);
END_ACTION

ACTION Wait_Arrive_action:
tonMoveDelay(IN:=TRUE , PT:= tMoveDelay);
END_ACTION

ACTION Wait_Arrive_exit:
tonMoveDelay(IN:=FALSE);
END_ACTION

ACTION Eject_action:
OEjector := TRUE;
tonEjectDelay(IN:=TRUE , PT:= tEjectorDelay);
END_ACTION

ACTION Eject_exit:
tonEjectDelay(IN:=FALSE);
END_ACTION

ACTION ResetEjector_action:
OEjector := FALSE;
tonEjectDelay(IN:=TRUE , PT:= tEjectorDelay);
END_ACTION

ACTION ResetEjector_exit:
tonEjectDelay(IN:=FALSE);
END_ACTION

ACTION ReturnToLoading_action:
fbDrive(
	bEnable:= TRUE,
	bStart:= TRUE,
	wTarget:= GPOS_LOADING);

tonMoveDelay(IN:=TRUE , PT:= tMoveDelay);
END_ACTION

ACTION ReturnToLoading_exit:
fbDrive(
	bStart:= FALSE);

tonMoveDelay(IN:=FALSE);
END_ACTION

ACTION Wait_Return_action:
tonMoveDelay(IN:=TRUE , PT:= tMoveDelay);
END_ACTION

ACTION Wait_Return_exit:
tonMoveDelay(IN:=FALSE);
END_ACTION

ACTION Done_action:
bDone := TRUE;
END_ACTION

ACTION Done_exit:
bDone := FALSE;
END_ACTION
END_PROGRAM

(* POU Processes/PRG_DeliverToGarbage2, SFC *)
PROGRAM PRG_DeliverToGarbage2
VAR_INPUT
	bExecute: BOOL;
END_VAR
VAR_INPUT
	bDone: BOOL;
END_VAR
VAR
	tonMoveDelay	: TON;
	tonEjectDelay	: TON;
	tMoveDelay	: TIME := T#3s;
	tEjectorDelay	: TIME := T#3s;
END_VAR
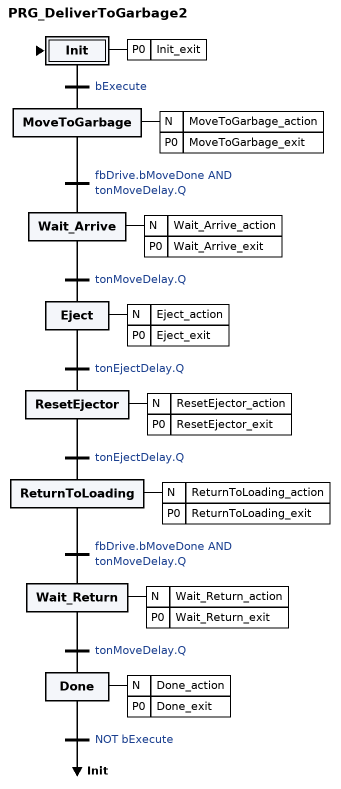
INITIAL_STEP Init:
	Init_exit(P0);
END_STEP
TRANSITION FROM Init TO MoveToGarbage := bExecute;
END_TRANSITION
STEP MoveToGarbage:
	MoveToGarbage_action(N);
	MoveToGarbage_exit(P0);
END_STEP
TRANSITION FROM MoveToGarbage TO Wait_Arrive := fbDrive.bMoveDone AND tonMoveDelay.Q;
END_TRANSITION
STEP Wait_Arrive:
	Wait_Arrive_action(N);
	Wait_Arrive_exit(P0);
END_STEP
TRANSITION FROM Wait_Arrive TO Eject := tonMoveDelay.Q;
END_TRANSITION
STEP Eject:
	Eject_action(N);
	Eject_exit(P0);
END_STEP
TRANSITION FROM Eject TO ResetEjector := tonEjectDelay.Q;
END_TRANSITION
STEP ResetEjector:
	ResetEjector_action(N);
	ResetEjector_exit(P0);
END_STEP
TRANSITION FROM ResetEjector TO ReturnToLoading := tonEjectDelay.Q;
END_TRANSITION
STEP ReturnToLoading:
	ReturnToLoading_action(N);
	ReturnToLoading_exit(P0);
END_STEP
TRANSITION FROM ReturnToLoading TO Wait_Return := fbDrive.bMoveDone AND tonMoveDelay.Q;
END_TRANSITION
STEP Wait_Return:
	Wait_Return_action(N);
	Wait_Return_exit(P0);
END_STEP
TRANSITION FROM Wait_Return TO Done := tonMoveDelay.Q;
END_TRANSITION
STEP Done:
	Done_action(N);
	Done_exit(P0);
END_STEP
TRANSITION FROM Done TO Init := NOT bExecute;
END_TRANSITION

ACTION Init_exit:
bDone := FALSE;
END_ACTION

ACTION MoveToGarbage_action:
fbDrive(
	bEnable:= TRUE,
	bStart:= TRUE,
	wTarget:= GPOS_GARBAGE);

tonMoveDelay(IN:=TRUE , PT:= tMoveDelay);
END_ACTION

ACTION MoveToGarbage_exit:
fbDrive(
	bStart:= FALSE);
tonMoveDelay(IN:=FALSE);
END_ACTION

ACTION Wait_Arrive_action:
tonMoveDelay(IN:=TRUE , PT:= tMoveDelay);
END_ACTION

ACTION Wait_Arrive_exit:
tonMoveDelay(IN:=FALSE);
END_ACTION

ACTION Eject_action:
OEjector := TRUE;
tonEjectDelay(IN:=TRUE , PT:= tEjectorDelay);
END_ACTION

ACTION Eject_exit:
tonEjectDelay(IN:=FALSE);
END_ACTION

ACTION ResetEjector_action:
OEjector := FALSE;
tonEjectDelay(IN:=TRUE , PT:= tEjectorDelay);
END_ACTION

ACTION ResetEjector_exit:
tonEjectDelay(IN:=FALSE);
END_ACTION

ACTION ReturnToLoading_action:
fbDrive(
	bEnable:= TRUE,
	bStart:= TRUE,
	wTarget:= GPOS_LOADING);

tonMoveDelay(IN:=TRUE , PT:= tMoveDelay);
END_ACTION

ACTION ReturnToLoading_exit:
fbDrive(
	bStart:= FALSE);

tonMoveDelay(IN:=FALSE);
END_ACTION

ACTION Wait_Return_action:
tonMoveDelay(IN:=TRUE , PT:= tMoveDelay);
END_ACTION

ACTION Wait_Return_exit:
tonMoveDelay(IN:=FALSE);
END_ACTION

ACTION Done_action:
bDone := TRUE;
END_ACTION

ACTION Done_exit:
bDone := FALSE;
END_ACTION
END_PROGRAM

(* POU Processes/PRG_ToColourSensor2, SFC *)
PROGRAM PRG_ToColourSensor2
VAR_INPUT
	bExecute: BOOL;
END_VAR
VAR_INPUT
	bDone: BOOL;
END_VAR
VAR
	tonMoveDelay	: TON;
	tonEjectDelay	: TON;
	tMoveDelay	: TIME := T#3s;
	tEjectorDelay	: TIME := T#3s;
END_VAR
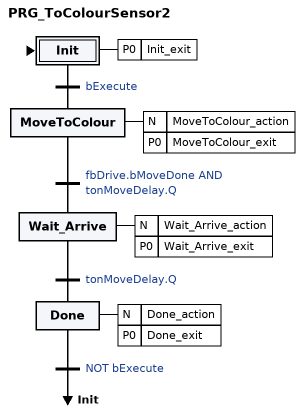
INITIAL_STEP Init:
	Init_exit(P0);
END_STEP
TRANSITION FROM Init TO MoveToColour := bExecute;
END_TRANSITION
STEP MoveToColour:
	MoveToColour_action(N);
	MoveToColour_exit(P0);
END_STEP
TRANSITION FROM MoveToColour TO Wait_Arrive := fbDrive.bMoveDone AND tonMoveDelay.Q;
END_TRANSITION
STEP Wait_Arrive:
	Wait_Arrive_action(N);
	Wait_Arrive_exit(P0);
END_STEP
TRANSITION FROM Wait_Arrive TO Done := tonMoveDelay.Q;
END_TRANSITION
STEP Done:
	Done_action(N);
	Done_exit(P0);
END_STEP
TRANSITION FROM Done TO Init := NOT bExecute;
END_TRANSITION

ACTION Init_exit:
bDone := FALSE;
END_ACTION

ACTION MoveToColour_action:
fbDrive(
	bEnable:= TRUE,
	bStart:= TRUE,
	wTarget:= GPOS_COLOR_SEN);

tonMoveDelay(IN:=TRUE , PT:= tMoveDelay);
END_ACTION

ACTION MoveToColour_exit:
fbDrive(
	bStart:= FALSE);
tonMoveDelay(IN:=FALSE);
END_ACTION

ACTION Wait_Arrive_action:
tonMoveDelay(IN:=TRUE , PT:= tMoveDelay);
END_ACTION

ACTION Wait_Arrive_exit:
tonMoveDelay(IN:=FALSE);
END_ACTION

ACTION Done_action:
bDone := TRUE;
END_ACTION

ACTION Done_exit:
bDone := FALSE;
END_ACTION
END_PROGRAM

(* POU Processes/PRG_DeliverToLow2, SFC *)
PROGRAM PRG_DeliverToLow2
VAR_INPUT
	bExecute: BOOL;
END_VAR
VAR_INPUT
	bDone: BOOL;
END_VAR
VAR
	tonMoveDelay	: TON;
	tonEjectDelay	: TON;
	tMoveDelay	: TIME := T#4s;
	tEjectorDelay	: TIME := T#3s;
END_VAR
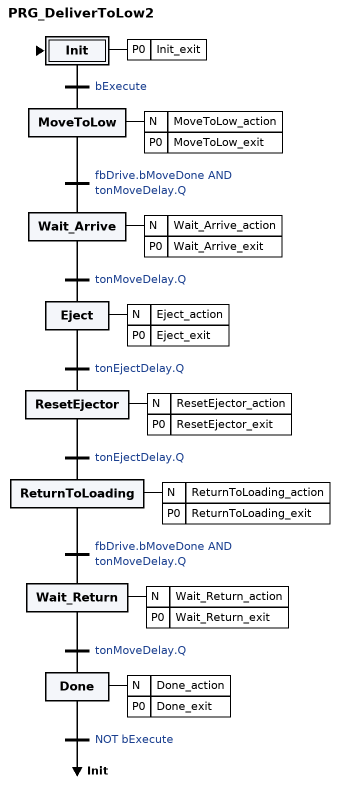
INITIAL_STEP Init:
	Init_exit(P0);
END_STEP
TRANSITION FROM Init TO MoveToLow := bExecute;
END_TRANSITION
STEP MoveToLow:
	MoveToLow_action(N);
	MoveToLow_exit(P0);
END_STEP
TRANSITION FROM MoveToLow TO Wait_Arrive := fbDrive.bMoveDone AND tonMoveDelay.Q;
END_TRANSITION
STEP Wait_Arrive:
	Wait_Arrive_action(N);
	Wait_Arrive_exit(P0);
END_STEP
TRANSITION FROM Wait_Arrive TO Eject := tonMoveDelay.Q;
END_TRANSITION
STEP Eject:
	Eject_action(N);
	Eject_exit(P0);
END_STEP
TRANSITION FROM Eject TO ResetEjector := tonEjectDelay.Q;
END_TRANSITION
STEP ResetEjector:
	ResetEjector_action(N);
	ResetEjector_exit(P0);
END_STEP
TRANSITION FROM ResetEjector TO ReturnToLoading := tonEjectDelay.Q;
END_TRANSITION
STEP ReturnToLoading:
	ReturnToLoading_action(N);
	ReturnToLoading_exit(P0);
END_STEP
TRANSITION FROM ReturnToLoading TO Wait_Return := fbDrive.bMoveDone AND tonMoveDelay.Q;
END_TRANSITION
STEP Wait_Return:
	Wait_Return_action(N);
	Wait_Return_exit(P0);
END_STEP
TRANSITION FROM Wait_Return TO Done := tonMoveDelay.Q;
END_TRANSITION
STEP Done:
	Done_action(N);
	Done_exit(P0);
END_STEP
TRANSITION FROM Done TO Init := NOT bExecute;
END_TRANSITION

ACTION Init_exit:
bDone := FALSE;
END_ACTION

ACTION MoveToLow_action:
tonMoveDelay(IN:=TRUE , PT:= tMoveDelay);
fbDrive(
	bEnable:= TRUE,
	bStart:= TRUE,
	wTarget:= GPOS_PIPE_LOW);
END_ACTION

ACTION MoveToLow_exit:
fbDrive(
	bStart:= FALSE);
tonMoveDelay(IN:=FALSE);
END_ACTION

ACTION Wait_Arrive_action:
tonMoveDelay(IN:=TRUE , PT:= tMoveDelay);
END_ACTION

ACTION Wait_Arrive_exit:
tonMoveDelay(IN:=FALSE);
END_ACTION

ACTION Eject_action:
OEjector := TRUE;
tonEjectDelay(IN:=TRUE , PT:= tEjectorDelay);
END_ACTION

ACTION Eject_exit:
tonEjectDelay(IN:=FALSE);
END_ACTION

ACTION ResetEjector_action:
OEjector := FALSE;
tonEjectDelay(IN:=TRUE , PT:= tEjectorDelay);
END_ACTION

ACTION ResetEjector_exit:
tonEjectDelay(IN:=FALSE);
END_ACTION

ACTION ReturnToLoading_action:
fbDrive(
	bEnable:= TRUE,
	bStart:= TRUE,
	wTarget:= GPOS_LOADING);

tonMoveDelay(IN:=TRUE , PT:= tMoveDelay);
END_ACTION

ACTION ReturnToLoading_exit:
fbDrive(
	bStart:= FALSE);

tonMoveDelay(IN:=FALSE);
END_ACTION

ACTION Wait_Return_action:
tonMoveDelay(IN:=TRUE , PT:= tMoveDelay);
END_ACTION

ACTION Wait_Return_exit:
tonMoveDelay(IN:=FALSE);
END_ACTION

ACTION Done_action:
bDone := TRUE;
END_ACTION

ACTION Done_exit:
bDone := FALSE;
END_ACTION
END_PROGRAM

(* POU Processes/PRG_DeliverToLow, SFC *)
PROGRAM PRG_DeliverToLow
VAR_INPUT
	bReset		: BOOL;	(*Reset program*)
	bExecute		: BOOL;	(*enable and run*)

END_VAR
VAR_OUTPUT
	bDone			: BOOL;
END_VAR
VAR
	tonMoveDelay	: TON;
	tonEjectDelay	: TON;
	SFCReset		: BOOL;

	tMoveDelay	: TIME := T#4s;
	tEjectorDelay	: TIME := T#3s;
END_VAR
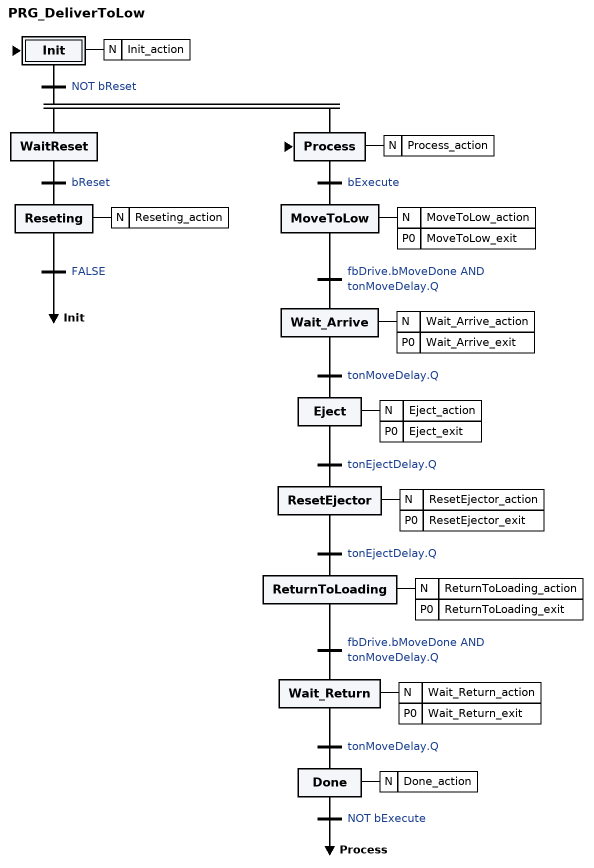
INITIAL_STEP Init:
	Init_action(N);
END_STEP
TRANSITION FROM Init TO (WaitReset, Process) := NOT bReset;
END_TRANSITION
STEP WaitReset:
END_STEP
TRANSITION FROM WaitReset TO Reseting := bReset;
END_TRANSITION
STEP Process:
	Process_action(N);
END_STEP
TRANSITION FROM Process TO MoveToLow := bExecute;
END_TRANSITION
STEP MoveToLow:
	MoveToLow_action(N);
	MoveToLow_exit(P0);
END_STEP
TRANSITION FROM MoveToLow TO Wait_Arrive := fbDrive.bMoveDone AND tonMoveDelay.Q;
END_TRANSITION
STEP Wait_Arrive:
	Wait_Arrive_action(N);
	Wait_Arrive_exit(P0);
END_STEP
TRANSITION FROM Wait_Arrive TO Eject := tonMoveDelay.Q;
END_TRANSITION
STEP Eject:
	Eject_action(N);
	Eject_exit(P0);
END_STEP
TRANSITION FROM Eject TO ResetEjector := tonEjectDelay.Q;
END_TRANSITION
STEP ResetEjector:
	ResetEjector_action(N);
	ResetEjector_exit(P0);
END_STEP
TRANSITION FROM ResetEjector TO ReturnToLoading := tonEjectDelay.Q;
END_TRANSITION
STEP ReturnToLoading:
	ReturnToLoading_action(N);
	ReturnToLoading_exit(P0);
END_STEP
TRANSITION FROM ReturnToLoading TO Wait_Return := fbDrive.bMoveDone AND tonMoveDelay.Q;
END_TRANSITION
STEP Wait_Return:
	Wait_Return_action(N);
	Wait_Return_exit(P0);
END_STEP
TRANSITION FROM Wait_Return TO Done := tonMoveDelay.Q;
END_TRANSITION
STEP Done:
	Done_action(N);
END_STEP
TRANSITION FROM Done TO Process := NOT bExecute;
END_TRANSITION
STEP Reseting:
	Reseting_action(N);
END_STEP
TRANSITION FROM Reseting TO Init := FALSE;
END_TRANSITION

ACTION Init_action:
SFCReset := FALSE;
bDone := FALSE;
END_ACTION

ACTION Process_action:
bDone := FALSE;
END_ACTION

ACTION MoveToLow_action:
bDone := FALSE;

fbDrive(
	bEnable:= TRUE,
	bStart:= TRUE,
	wTarget:= GPOS_PIPE_LOW);

tonMoveDelay(IN:=TRUE , PT:= tMoveDelay);
END_ACTION

ACTION MoveToLow_exit:
fbDrive(
	bStart:= FALSE);
tonMoveDelay(IN:=FALSE);
END_ACTION

ACTION Wait_Arrive_action:
tonMoveDelay(IN:=TRUE , PT:= tMoveDelay);
END_ACTION

ACTION Wait_Arrive_exit:
tonMoveDelay(IN:=FALSE);
END_ACTION

ACTION Eject_action:
OEjector := TRUE;
tonEjectDelay(IN:=TRUE , PT:= tEjectorDelay);
END_ACTION

ACTION Eject_exit:
tonEjectDelay(IN:=FALSE);
END_ACTION

ACTION ResetEjector_action:
OEjector := FALSE;
tonEjectDelay(IN:=TRUE , PT:= tEjectorDelay);
END_ACTION

ACTION ResetEjector_exit:
tonEjectDelay(IN:=FALSE);
END_ACTION

ACTION ReturnToLoading_action:
fbDrive(
	bEnable:= TRUE,
	bStart:= TRUE,
	wTarget:= GPOS_LOADING);

tonMoveDelay(IN:=TRUE , PT:= tMoveDelay);
END_ACTION

ACTION ReturnToLoading_exit:
fbDrive(
	bStart:= FALSE);

tonMoveDelay(IN:=FALSE);
END_ACTION

ACTION Wait_Return_action:
tonMoveDelay(IN:=TRUE , PT:= tMoveDelay);
END_ACTION

ACTION Wait_Return_exit:
tonMoveDelay(IN:=FALSE);
END_ACTION

ACTION Done_action:
bDone := TRUE;
END_ACTION

ACTION Reseting_action:
SFCReset := TRUE;
END_ACTION
END_PROGRAM

(* POU Processes/PRG_DeliverToGarbage, SFC *)
PROGRAM PRG_DeliverToGarbage
VAR_INPUT
	bReset		: BOOL;	(*Reset program*)
	bExecute		: BOOL;	(*enable and run*)
END_VAR
VAR_OUTPUT
	bDone			: BOOL;
END_VAR
VAR
	tonMoveDelay	: TON;
	tonEjectDelay	: TON;
	SFCReset		: BOOL;

	tMoveDelay	: TIME := T#4s;
	tEjectorDelay	: TIME := T#2s;
END_VAR
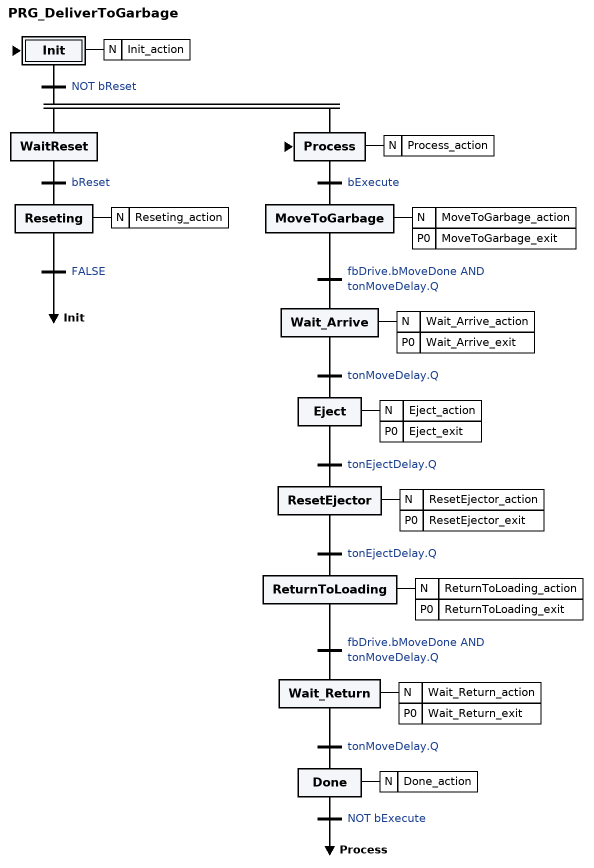
INITIAL_STEP Init:
	Init_action(N);
END_STEP
TRANSITION FROM Init TO (WaitReset, Process) := NOT bReset;
END_TRANSITION
STEP WaitReset:
END_STEP
TRANSITION FROM WaitReset TO Reseting := bReset;
END_TRANSITION
STEP Process:
	Process_action(N);
END_STEP
TRANSITION FROM Process TO MoveToGarbage := bExecute;
END_TRANSITION
STEP MoveToGarbage:
	MoveToGarbage_action(N);
	MoveToGarbage_exit(P0);
END_STEP
TRANSITION FROM MoveToGarbage TO Wait_Arrive := fbDrive.bMoveDone AND tonMoveDelay.Q;
END_TRANSITION
STEP Wait_Arrive:
	Wait_Arrive_action(N);
	Wait_Arrive_exit(P0);
END_STEP
TRANSITION FROM Wait_Arrive TO Eject := tonMoveDelay.Q;
END_TRANSITION
STEP Eject:
	Eject_action(N);
	Eject_exit(P0);
END_STEP
TRANSITION FROM Eject TO ResetEjector := tonEjectDelay.Q;
END_TRANSITION
STEP ResetEjector:
	ResetEjector_action(N);
	ResetEjector_exit(P0);
END_STEP
TRANSITION FROM ResetEjector TO ReturnToLoading := tonEjectDelay.Q;
END_TRANSITION
STEP ReturnToLoading:
	ReturnToLoading_action(N);
	ReturnToLoading_exit(P0);
END_STEP
TRANSITION FROM ReturnToLoading TO Wait_Return := fbDrive.bMoveDone AND tonMoveDelay.Q;
END_TRANSITION
STEP Wait_Return:
	Wait_Return_action(N);
	Wait_Return_exit(P0);
END_STEP
TRANSITION FROM Wait_Return TO Done := tonMoveDelay.Q;
END_TRANSITION
STEP Done:
	Done_action(N);
END_STEP
TRANSITION FROM Done TO Process := NOT bExecute;
END_TRANSITION
STEP Reseting:
	Reseting_action(N);
END_STEP
TRANSITION FROM Reseting TO Init := FALSE;
END_TRANSITION

ACTION Init_action:
SFCReset := FALSE;
bDone := FALSE;
END_ACTION

ACTION Process_action:
bDone := FALSE;
END_ACTION

ACTION MoveToGarbage_action:
bDone := FALSE;

fbDrive(
	bEnable:= TRUE,
	bStart:= TRUE,
	wTarget:= GPOS_GARBAGE);

tonMoveDelay(IN:=TRUE , PT:= tMoveDelay);
END_ACTION

ACTION MoveToGarbage_exit:
fbDrive(
	bStart:= FALSE);

tonMoveDelay(IN:=FALSE);
END_ACTION

ACTION Wait_Arrive_action:
tonMoveDelay(IN:=TRUE , PT:= tMoveDelay);
END_ACTION

ACTION Wait_Arrive_exit:
tonMoveDelay(IN:=FALSE);
END_ACTION

ACTION Eject_action:
OEjector := TRUE;
tonEjectDelay(IN:=TRUE , PT:= tEjectorDelay);
END_ACTION

ACTION Eject_exit:
tonEjectDelay(IN:=FALSE);
END_ACTION

ACTION ResetEjector_action:
OEjector := FALSE;
tonEjectDelay(IN:=TRUE , PT:= tEjectorDelay);
END_ACTION

ACTION ResetEjector_exit:
tonEjectDelay(IN:=FALSE);
END_ACTION

ACTION ReturnToLoading_action:
fbDrive(
	bEnable:= TRUE,
	bStart:= TRUE,
	wTarget:= GPOS_LOADING);

tonMoveDelay(IN:=TRUE , PT:= tMoveDelay);
END_ACTION

ACTION ReturnToLoading_exit:
fbDrive(
	bStart:= FALSE);

tonMoveDelay(IN:=FALSE);
END_ACTION

ACTION Wait_Return_action:
tonMoveDelay(IN:=TRUE , PT:= tMoveDelay);
END_ACTION

ACTION Wait_Return_exit:
tonMoveDelay(IN:=FALSE);
END_ACTION

ACTION Done_action:
bDone := TRUE;
END_ACTION

ACTION Reseting_action:
SFCReset := TRUE;
END_ACTION
END_PROGRAM

(* POU Processes/PRG_DeliverToMid, SFC *)
PROGRAM PRG_DeliverToMid
VAR_INPUT
	bReset		: BOOL;	(*Reset program*)
	bExecute		: BOOL;	(*enable and run*)
END_VAR
VAR_OUTPUT
	bDone			: BOOL;
END_VAR
VAR
	tonMoveDelay	: TON;
	tonEjectDelay	: TON;
	SFCReset		: BOOL;

	tMoveDelay	: TIME := T#4s;
	tEjectorDelay	: TIME := T#2s;
END_VAR
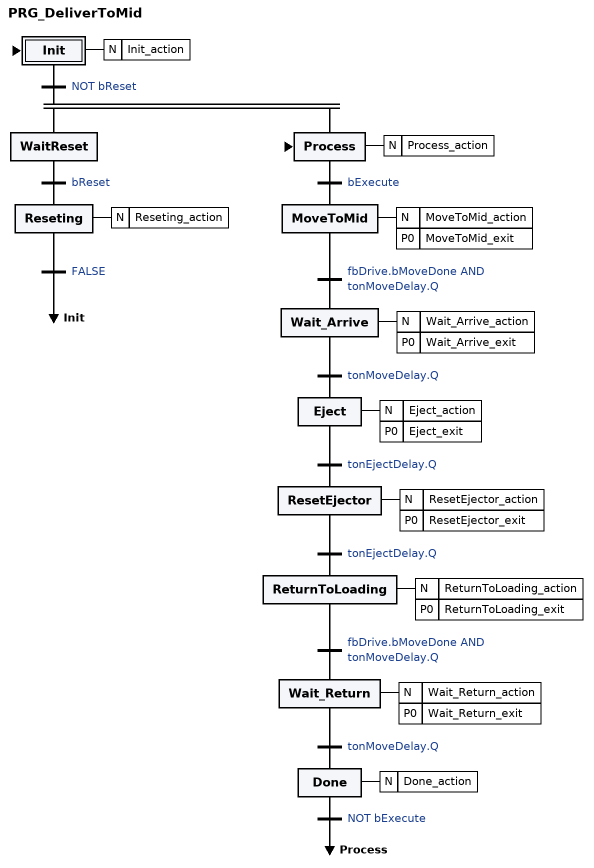
INITIAL_STEP Init:
	Init_action(N);
END_STEP
TRANSITION FROM Init TO (WaitReset, Process) := NOT bReset;
END_TRANSITION
STEP WaitReset:
END_STEP
TRANSITION FROM WaitReset TO Reseting := bReset;
END_TRANSITION
STEP Process:
	Process_action(N);
END_STEP
TRANSITION FROM Process TO MoveToMid := bExecute;
END_TRANSITION
STEP MoveToMid:
	MoveToMid_action(N);
	MoveToMid_exit(P0);
END_STEP
TRANSITION FROM MoveToMid TO Wait_Arrive := fbDrive.bMoveDone AND tonMoveDelay.Q;
END_TRANSITION
STEP Wait_Arrive:
	Wait_Arrive_action(N);
	Wait_Arrive_exit(P0);
END_STEP
TRANSITION FROM Wait_Arrive TO Eject := tonMoveDelay.Q;
END_TRANSITION
STEP Eject:
	Eject_action(N);
	Eject_exit(P0);
END_STEP
TRANSITION FROM Eject TO ResetEjector := tonEjectDelay.Q;
END_TRANSITION
STEP ResetEjector:
	ResetEjector_action(N);
	ResetEjector_exit(P0);
END_STEP
TRANSITION FROM ResetEjector TO ReturnToLoading := tonEjectDelay.Q;
END_TRANSITION
STEP ReturnToLoading:
	ReturnToLoading_action(N);
	ReturnToLoading_exit(P0);
END_STEP
TRANSITION FROM ReturnToLoading TO Wait_Return := fbDrive.bMoveDone AND tonMoveDelay.Q;
END_TRANSITION
STEP Wait_Return:
	Wait_Return_action(N);
	Wait_Return_exit(P0);
END_STEP
TRANSITION FROM Wait_Return TO Done := tonMoveDelay.Q;
END_TRANSITION
STEP Done:
	Done_action(N);
END_STEP
TRANSITION FROM Done TO Process := NOT bExecute;
END_TRANSITION
STEP Reseting:
	Reseting_action(N);
END_STEP
TRANSITION FROM Reseting TO Init := FALSE;
END_TRANSITION

ACTION Init_action:
SFCReset := FALSE;
bDone := FALSE;
END_ACTION

ACTION Process_action:
bDone := FALSE;
END_ACTION

ACTION MoveToMid_action:
bDone := FALSE;

fbDrive(
	bEnable:= TRUE,
	bStart:= TRUE,
	wTarget:=GPOS_PIPE_MID);

tonMoveDelay(IN:=TRUE , PT:= tMoveDelay);
END_ACTION

ACTION MoveToMid_exit:
fbDrive(
	bStart:= FALSE);

tonMoveDelay(IN:=FALSE);
END_ACTION

ACTION Wait_Arrive_action:
tonMoveDelay(IN:=TRUE , PT:= tMoveDelay);
END_ACTION

ACTION Wait_Arrive_exit:
tonMoveDelay(IN:=FALSE);
END_ACTION

ACTION Eject_action:
OEjector := TRUE;
tonEjectDelay(IN:=TRUE , PT:= tEjectorDelay);
END_ACTION

ACTION Eject_exit:
tonEjectDelay(IN:=FALSE);
END_ACTION

ACTION ResetEjector_action:
OEjector := FALSE;
tonEjectDelay(IN:=TRUE , PT:= tEjectorDelay);
END_ACTION

ACTION ResetEjector_exit:
tonEjectDelay(IN:=FALSE);
END_ACTION

ACTION ReturnToLoading_action:
fbDrive(
	bEnable:= TRUE,
	bStart:= TRUE,
	wTarget:= GPOS_LOADING);

tonMoveDelay(IN:=TRUE , PT:= tMoveDelay);
END_ACTION

ACTION ReturnToLoading_exit:
fbDrive(
	bStart:= FALSE);

tonMoveDelay(IN:=FALSE);
END_ACTION

ACTION Wait_Return_action:
tonMoveDelay(IN:=TRUE , PT:= tMoveDelay);
END_ACTION

ACTION Wait_Return_exit:
tonMoveDelay(IN:=FALSE);
END_ACTION

ACTION Done_action:
bDone := TRUE;
END_ACTION

ACTION Reseting_action:
SFCReset := TRUE;
END_ACTION
END_PROGRAM

(* POU Processes/PRG_DeliverToUp, SFC *)
PROGRAM PRG_DeliverToUp
VAR_INPUT
	bReset		: BOOL;	(*Reset program*)
	bExecute		: BOOL;	(*enable and run*)
END_VAR
VAR_OUTPUT
	bDone			: BOOL;
END_VAR
VAR
	tonMoveDelay	: TON;
	tonEjectDelay	: TON;
	SFCReset		: BOOL;

	tMoveDelay	: TIME := T#4s;
	tEjectorDelay	: TIME := T#2s;
END_VAR
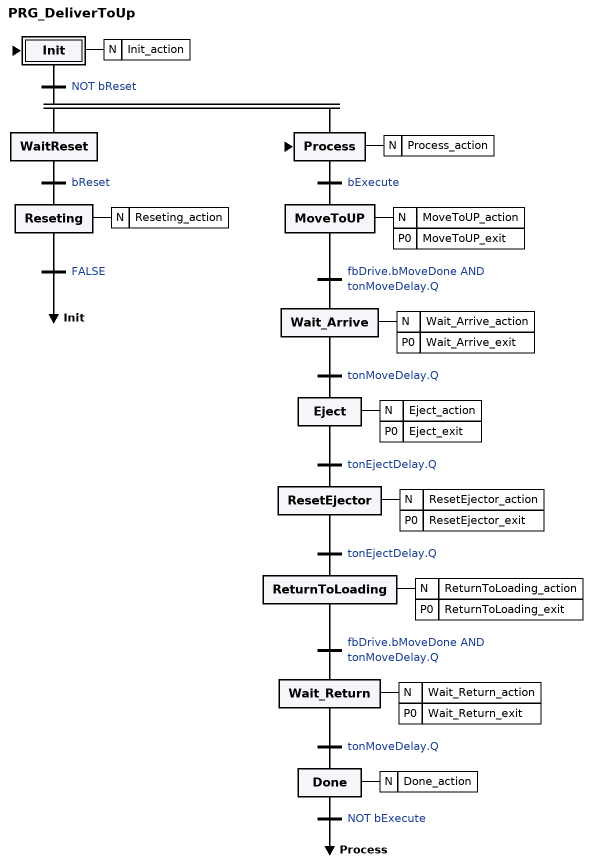
INITIAL_STEP Init:
	Init_action(N);
END_STEP
TRANSITION FROM Init TO (WaitReset, Process) := NOT bReset;
END_TRANSITION
STEP WaitReset:
END_STEP
TRANSITION FROM WaitReset TO Reseting := bReset;
END_TRANSITION
STEP Process:
	Process_action(N);
END_STEP
TRANSITION FROM Process TO MoveToUP := bExecute;
END_TRANSITION
STEP MoveToUP:
	MoveToUP_action(N);
	MoveToUP_exit(P0);
END_STEP
TRANSITION FROM MoveToUP TO Wait_Arrive := fbDrive.bMoveDone AND tonMoveDelay.Q;
END_TRANSITION
STEP Wait_Arrive:
	Wait_Arrive_action(N);
	Wait_Arrive_exit(P0);
END_STEP
TRANSITION FROM Wait_Arrive TO Eject := tonMoveDelay.Q;
END_TRANSITION
STEP Eject:
	Eject_action(N);
	Eject_exit(P0);
END_STEP
TRANSITION FROM Eject TO ResetEjector := tonEjectDelay.Q;
END_TRANSITION
STEP ResetEjector:
	ResetEjector_action(N);
	ResetEjector_exit(P0);
END_STEP
TRANSITION FROM ResetEjector TO ReturnToLoading := tonEjectDelay.Q;
END_TRANSITION
STEP ReturnToLoading:
	ReturnToLoading_action(N);
	ReturnToLoading_exit(P0);
END_STEP
TRANSITION FROM ReturnToLoading TO Wait_Return := fbDrive.bMoveDone AND tonMoveDelay.Q;
END_TRANSITION
STEP Wait_Return:
	Wait_Return_action(N);
	Wait_Return_exit(P0);
END_STEP
TRANSITION FROM Wait_Return TO Done := tonMoveDelay.Q;
END_TRANSITION
STEP Done:
	Done_action(N);
END_STEP
TRANSITION FROM Done TO Process := NOT bExecute;
END_TRANSITION
STEP Reseting:
	Reseting_action(N);
END_STEP
TRANSITION FROM Reseting TO Init := FALSE;
END_TRANSITION

ACTION Init_action:
SFCReset := FALSE;
bDone := FALSE;
END_ACTION

ACTION Process_action:
bDone := FALSE;
END_ACTION

ACTION MoveToUP_action:
bDone := FALSE;

fbDrive(
	bEnable:= TRUE,
	bStart:= TRUE,
	wTarget:= GPOS_PIPE_UP);

tonMoveDelay(IN:=TRUE , PT:= tMoveDelay);
END_ACTION

ACTION MoveToUP_exit:
fbDrive(
	bStart:= FALSE);

tonMoveDelay(IN:=FALSE);
END_ACTION

ACTION Wait_Arrive_action:
tonMoveDelay(IN:=TRUE , PT:= tMoveDelay);
END_ACTION

ACTION Wait_Arrive_exit:
tonMoveDelay(IN:=FALSE);
END_ACTION

ACTION Eject_action:
OEjector := TRUE;
tonEjectDelay(IN:=TRUE , PT:= tEjectorDelay);
END_ACTION

ACTION Eject_exit:
tonEjectDelay(IN:=FALSE);
END_ACTION

ACTION ResetEjector_action:
OEjector := FALSE;
tonEjectDelay(IN:=TRUE , PT:= tEjectorDelay);
END_ACTION

ACTION ResetEjector_exit:
tonEjectDelay(IN:=FALSE);
END_ACTION

ACTION ReturnToLoading_action:
fbDrive(
	bEnable:= TRUE,
	bStart:= TRUE,
	wTarget:= GPOS_LOADING);

tonMoveDelay(IN:=TRUE , PT:= tMoveDelay);
END_ACTION

ACTION ReturnToLoading_exit:
fbDrive(
	bStart:= FALSE);

tonMoveDelay(IN:=FALSE);
END_ACTION

ACTION Wait_Return_action:
tonMoveDelay(IN:=TRUE , PT:= tMoveDelay);
END_ACTION

ACTION Wait_Return_exit:
tonMoveDelay(IN:=FALSE);
END_ACTION

ACTION Done_action:
bDone := TRUE;
END_ACTION

ACTION Reseting_action:
SFCReset := TRUE;
END_ACTION
END_PROGRAM

(* POU Processes/PRG_ToColourSensor, SFC *)
PROGRAM PRG_ToColourSensor
VAR_INPUT
	bReset		: BOOL;	(*Reset program*)
	bExecute		: BOOL;	(*enable and run*)
END_VAR
VAR_OUTPUT
	bDone			: BOOL;
END_VAR
VAR

	tonMoveDelay	: TON;
	SFCReset		: BOOL;
	tMoveDelay	: TIME := T#4s;
END_VAR
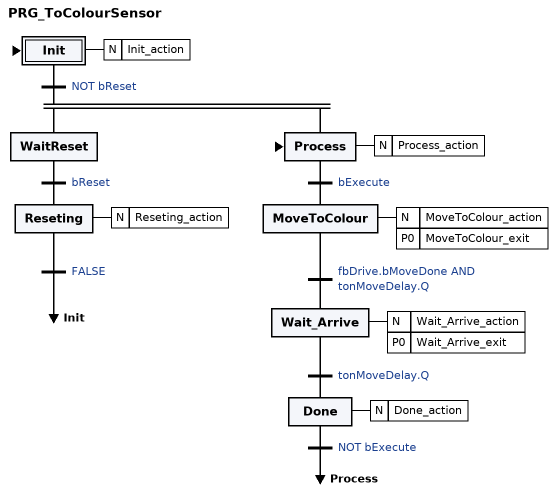
INITIAL_STEP Init:
	Init_action(N);
END_STEP
TRANSITION FROM Init TO (WaitReset, Process) := NOT bReset;
END_TRANSITION
STEP WaitReset:
END_STEP
TRANSITION FROM WaitReset TO Reseting := bReset;
END_TRANSITION
STEP Process:
	Process_action(N);
END_STEP
TRANSITION FROM Process TO MoveToColour := bExecute;
END_TRANSITION
STEP MoveToColour:
	MoveToColour_action(N);
	MoveToColour_exit(P0);
END_STEP
TRANSITION FROM MoveToColour TO Wait_Arrive := fbDrive.bMoveDone AND tonMoveDelay.Q;
END_TRANSITION
STEP Wait_Arrive:
	Wait_Arrive_action(N);
	Wait_Arrive_exit(P0);
END_STEP
TRANSITION FROM Wait_Arrive TO Done := tonMoveDelay.Q;
END_TRANSITION
STEP Done:
	Done_action(N);
END_STEP
TRANSITION FROM Done TO Process := NOT bExecute;
END_TRANSITION
STEP Reseting:
	Reseting_action(N);
END_STEP
TRANSITION FROM Reseting TO Init := FALSE;
END_TRANSITION

ACTION Init_action:
SFCReset := FALSE;
bDone := FALSE;
END_ACTION

ACTION Process_action:
bDone := FALSE;
END_ACTION

ACTION MoveToColour_action:
bDone := FALSE;

fbDrive(
	bEnable:= TRUE,
	bStart:= TRUE,
	wTarget:= GPOS_COLOR_SEN);

tonMoveDelay(IN:=TRUE , PT:= tMoveDelay);

(*
tonMoveDelay(IN:=TRUE , PT:= tMoveDelay);
*)
END_ACTION

ACTION MoveToColour_exit:
fbDrive(
	bStart:= FALSE);

tonMoveDelay(IN:=FALSE);
END_ACTION

ACTION Wait_Arrive_action:
tonMoveDelay(IN:=TRUE , PT:= tMoveDelay);
END_ACTION

ACTION Wait_Arrive_exit:
tonMoveDelay(IN:=FALSE);
END_ACTION

ACTION Done_action:
bDone := TRUE;
END_ACTION

ACTION Reseting_action:
SFCReset := TRUE;
END_ACTION
END_PROGRAM
